// TIA Portal project "Depo Seviye Kontrolü" (V17)

(* hardware
DEVICE "S71500/ET200MP-Station_1"  S7-1500 station
   slot 0: "Profilschiene_0"  6ES7 590-1***0-0AA0
   slot 1: "PLC_1"  CPU 1511-1 PN  6ES7 511-1AK00-0AB0  V1.8
   slot 2: "AI 8xU/I/RTD/TC ST_1"  AI 8xU/I/RTD/TC ST  6ES7 531-7KF00-0AB0  V2.0
   slot 3: "AI 8xU/I/RTD/TC ST_2"  AI 8xU/I/RTD/TC ST  6ES7 531-7KF00-0AB0  V2.0
   slot 4: "AI 8xU/I/RTD/TC ST_3"  AI 8xU/I/RTD/TC ST  6ES7 531-7KF00-0AB0  V2.0
   slot 5: "AI 8xU/I/RTD/TC ST_4"  AI 8xU/I/RTD/TC ST  6ES7 531-7KF00-0AB0  V2.0
   slot 6: "DI 16x24VDC BA_1"  DI 16x24VDC BA  6ES7 521-1BH10-0AA0  V1.0
*)

// ===== PLC "PLC_1"  CPU 1511-1 PN =====

VAR_GLOBAL   // PLC tag table "Standard-Variablentabelle"
   "START" AT %E0.0 : Bool;
   "1.POMPA" AT %A0.0 : Bool;
   "S1 SENSÖRÜ" AT %E0.1 : Bool;
   "YARDIMCI KONTAK" AT %M0.0 : Bool;
   "S2 SENSÖRÜ" AT %I0.2 : Bool;
   "2.POMPA" AT %Q0.1 : Bool;
   "UYARI IŞIĞI" AT %Q0.2 : Bool;
   "ACİL STOP" AT %I0.3 : Bool;
   "SESLİ İKAZ" AT %Q0.3 : Bool;
END_VAR

FUNCTION "MHJ-PLC-Lab-Function-S71500" : Void   // FC9000, SCL
{ S7_Optimized_Access := 'TRUE' }
VERSION : 0.1
   VAR_TEMP
      Value : Byte;
      ForCounter : Int;
   END_VAR
   VAR CONSTANT
      Value_01_DW : DWord := 16#1223_5486;
      Value_02_DW : DWord := 16#A6C9_D1F5;
   END_VAR
BEGIN

   #Value:=PEEK(area := 16#82,
        dbNumber := 0,
        byteOffset := 511);
   #Value := #Value + 1;

   POKE(area := 16#82,
        dbNumber := 0,
        byteOffset := 511,
        value := #Value);

   POKE(area := 16#82,
        dbNumber := 0,
        byteOffset := 1016,
        value := #Value_01_DW);
   POKE(area := 16#82,
        dbNumber := 0,
        byteOffset := 1020,
        value := #Value_02_DW);

   FOR #ForCounter := 0 TO 63 DO
       #Value:=PEEK(area := 16#1,
            dbNumber := 0,
            byteOffset := #ForCounter);
       POKE(area := 16#81,
            dbNumber := 0,
            byteOffset := #ForCounter,
            value := #Value);
   END_FOR;
   #Value := PEEK(area := 16#1,
                  dbNumber := 0,
                  byteOffset := 512);
   POKE(area := 16#82,
        dbNumber := 0,
        byteOffset := 512,
        value := #Value);
END_FUNCTION

ORGANIZATION_BLOCK "Main"   // OB1, LAD, ProgramCycle
TITLE = "Main Program Sweep (Cycle)"
{ S7_Optimized_Access := 'TRUE' }
VERSION : 0.1
   VAR_INPUT
      Initial_Call : Bool;   // Initial call of this OB
      Remanence : Bool;   // =True, if remanent data are available
   END_VAR
   VAR_TEMP   // added for the SCL form of the ladder/FBD networks
      _w1 : Bool;
   END_VAR
BEGIN

REGION Network 1
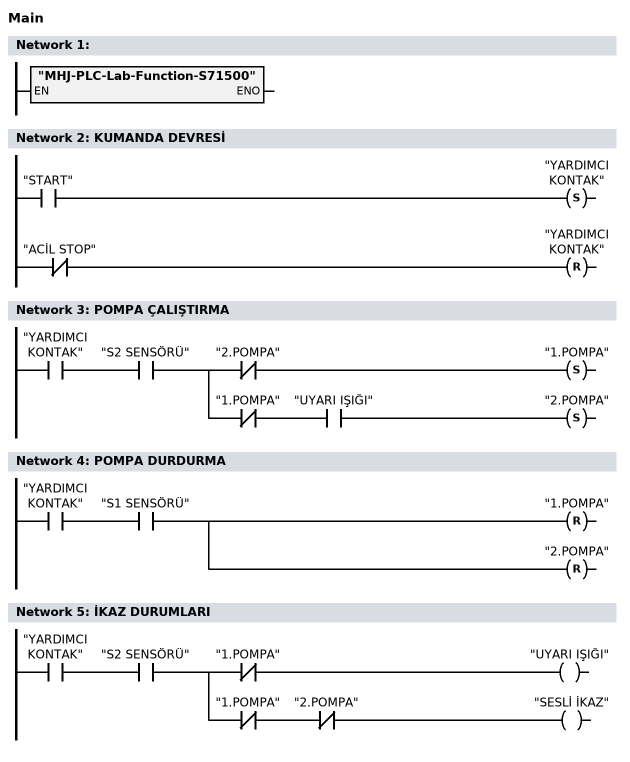
   RUNG wire#powerrail
      "MHJ-PLC-Lab-Function-S71500"()
   END_RUNG
   // the same network as SCL:
   "MHJ-PLC-Lab-Function-S71500"();
END_REGION

REGION Network 2: KUMANDA DEVRESİ
   RUNG wire#powerrail
      Contact( "START" )
      S_Coil( "YARDIMCI KONTAK" )
   END_RUNG
   RUNG wire#powerrail
      I_Contact( "ACİL STOP" )
      R_Coil( "YARDIMCI KONTAK" )
   END_RUNG
   // the same network as SCL:
   IF "START" THEN "YARDIMCI KONTAK" := TRUE; END_IF;
   IF NOT "ACİL STOP" THEN "YARDIMCI KONTAK" := FALSE; END_IF;
END_REGION

REGION Network 3: POMPA ÇALIŞTIRMA
   RUNG wire#powerrail
      Contact( "YARDIMCI KONTAK" )
      Contact( "S2 SENSÖRÜ" )
      wire#w1
      I_Contact( "2.POMPA" )
      S_Coil( "1.POMPA" )
   END_RUNG
   RUNG wire#w1
      I_Contact( "1.POMPA" )
      Contact( "UYARI IŞIĞI" )
      S_Coil( "2.POMPA" )
   END_RUNG
   // the same network as SCL:
   #_w1 := "YARDIMCI KONTAK" AND "S2 SENSÖRÜ";
   IF #_w1 AND NOT "2.POMPA" THEN "1.POMPA" := TRUE; END_IF;
   IF #_w1 AND NOT "1.POMPA" AND "UYARI IŞIĞI" THEN "2.POMPA" := TRUE; END_IF;
END_REGION

REGION Network 4: POMPA DURDURMA
   RUNG wire#powerrail
      Contact( "YARDIMCI KONTAK" )
      Contact( "S1 SENSÖRÜ" )
      wire#w1
      R_Coil( "1.POMPA" )
   END_RUNG
   RUNG wire#w1
      R_Coil( "2.POMPA" )
   END_RUNG
   // the same network as SCL:
   IF "YARDIMCI KONTAK" AND "S1 SENSÖRÜ" THEN
       "1.POMPA" := FALSE;
       "2.POMPA" := FALSE;
   END_IF;
END_REGION

REGION Network 5: İKAZ DURUMLARI
   RUNG wire#powerrail
      Contact( "YARDIMCI KONTAK" )
      Contact( "S2 SENSÖRÜ" )
      wire#w1
      I_Contact( "1.POMPA" )
      Coil( "UYARI IŞIĞI" )
   END_RUNG
   RUNG wire#w1
      I_Contact( "1.POMPA" )
      I_Contact( "2.POMPA" )
      Coil( "SESLİ İKAZ" )
   END_RUNG
   // the same network as SCL:
   #_w1 := "YARDIMCI KONTAK" AND "S2 SENSÖRÜ";
   "UYARI IŞIĞI" := #_w1 AND NOT "1.POMPA";
   "SESLİ İKAZ" := #_w1 AND NOT "1.POMPA" AND NOT "2.POMPA";
END_REGION
END_ORGANIZATION_BLOCK